# EPICS substitutions: Neslab.substitutions
file Neslab.template
{
pattern {S}
        {CG3:SE:NESLAB}
}
